FUNCTION_BLOCK SENSOR_DETECTOR
  {SET_ATTRIBUTE(OpcUa, SERVICE)}
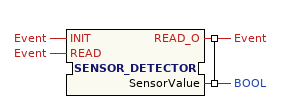
  EVENT_INPUT
    INIT;
    READ;
  END_EVENT
  EVENT_OUTPUT
    READ_O WITH SensorValue;
  END_EVENT
  VAR_OUTPUT
    SensorValue : BOOL;
  END_VAR
END_FUNCTION_BLOCK
